(* CODESYS project cds

Project tree, tasks and I/O mapping:
  Device : CODESYS Control RTE V3 x64, CODESYS, version 3.5.21.0
    application Application
      libraries: Standard, 3.5.18.0 (System)
      task MainTask (cyclic, interval t#20ms, priority 1) calls PLC_PRG
      program PLC_PRG [ST]
*)

// Device/Application/PLC_PRG
PROGRAM PLC_PRG
VAR
	x :bool;
END_VAR

x := not x;

END_PROGRAM
